FUNCTION_BLOCK FB_RecipeFactory_Test EXTENDS TcUnit.FB_TestSuite
VAR
    Factory : FB_RecipeFactory;
    Config  : ST_RecipeBuilder_Config;
END_VAR

Test_InjectsConfigProviderToAllBuilders();
Test_ReturnsCorrectBuilder();
Test_ReturnsZeroOnInvalidID();
Test_UpdatesConfigForAllBuilders();

METHOD Test_InjectsConfigProviderToAllBuilders
VAR_INST
    MockProvider : FB_MockConfigProvider;
END_VAR
VAR
    TestConfig       : ST_RecipeBuilder_Config;
    BuilderWings     : I_RecipeBuilder;
    BuilderFlaps     : I_RecipeBuilder;
    BuilderArona     : I_RecipeBuilder;
    BuilderCircle    : I_RecipeBuilder;
    BuilderRectangle : I_RecipeBuilder;
    
    iMockProvider    : I_GantryConfigProvider;
END_VAR
TEST('Test_InjectsConfigProviderToAllBuilders');

// 1. ARRANGE
// Rzutujemy instancję bloku na interfejs (aby kompilator wiedział, jak je porównywać)
iMockProvider := MockProvider;

// 2. ACT
Factory.InitializeFactory(Config := TestConfig, ConfigProvider := iMockProvider);

// Wyciągamy instancje z fabryki
BuilderWings     := Factory.GetBuilder(E_RecipeID.ePTPBorgoWings);
BuilderFlaps     := Factory.GetBuilder(E_RecipeID.ePTPBorgoFlaps);
BuilderArona     := Factory.GetBuilder(E_RecipeID.ePTPArona);
BuilderCircle    := Factory.GetBuilder(E_RecipeID.eNCICircle);
BuilderRectangle := Factory.GetBuilder(E_RecipeID.ePTPRectangle);

// 3. ASSERT
AssertTrue(Condition := (BuilderWings.ConfigProvider = iMockProvider),
           Message := 'BuilderWings nie otrzymal wstrzyknietego ConfigProvidera!');
AssertTrue(Condition := (BuilderFlaps.ConfigProvider = iMockProvider),
           Message := 'BuilderFlaps nie otrzymal wstrzyknietego ConfigProvidera!');
AssertTrue(Condition := (BuilderArona.ConfigProvider = iMockProvider),
           Message := 'BuilderArona nie otrzymal wstrzyknietego ConfigProvidera!');
AssertTrue(Condition := (BuilderCircle.ConfigProvider = iMockProvider),
           Message := 'BuilderCircle nie otrzymal wstrzyknietego ConfigProvidera!');
AssertTrue(Condition := (BuilderRectangle.ConfigProvider = iMockProvider),
           Message := 'BuilderRectangle nie otrzymal wstrzyknietego ConfigProvidera!');

TEST_FINISHED();
END_METHOD

METHOD Test_ReturnsCorrectBuilder
VAR
    BuilderWings     : I_RecipeBuilder;
    BuilderFlaps     : I_RecipeBuilder;
    BuilderArona     : I_RecipeBuilder;
    BuilderCircle    : I_RecipeBuilder; // Dodane!
    BuilderRectangle : I_RecipeBuilder; // Dodane!
END_VAR
TEST('Test_ReturnsCorrectBuilder');

// 1. ACT - Prosimy fabrykę o wszystkie wspierane przepisy
BuilderWings     := Factory.GetBuilder(E_RecipeID.ePTPBorgoWings);
BuilderFlaps     := Factory.GetBuilder(E_RecipeID.ePTPBorgoFlaps);
BuilderArona     := Factory.GetBuilder(E_RecipeID.ePTPArona);
BuilderCircle    := Factory.GetBuilder(E_RecipeID.eNCICircle);
BuilderRectangle := Factory.GetBuilder(E_RecipeID.ePTPRectangle);

// 2. ASSERT - Sprawdzamy, czy żaden z nich nie jest pusty (0)
AssertTrue(Condition := (BuilderWings <> 0), Message := 'Fabryka zwrocila 0 dla eBorgoWings!');
AssertTrue(Condition := (BuilderFlaps <> 0), Message := 'Fabryka zwrocila 0 dla eBorgoFlaps!');
AssertTrue(Condition := (BuilderArona <> 0), Message := 'Fabryka zwrocila 0 dla eArona!');
AssertTrue(Condition := (BuilderCircle <> 0), Message := 'Fabryka zwrocila 0 dla eCircle!');
AssertTrue(Condition := (BuilderRectangle <> 0), Message := 'Fabryka zwrocila 0 dla eRectangle!');

TEST_FINISHED();
END_METHOD

METHOD Test_ReturnsZeroOnInvalidID
VAR
    ReturnedBuilder : I_RecipeBuilder;
END_VAR


TEST('Test_ReturnsZeroOnInvalidID');

// Act - prosimy o eNone (ekran powitalny, bez wybranego programu)
ReturnedBuilder := Factory.GetBuilder(E_RecipeID.eNone);

// Assert - fabryka musi zwrócić 0
AssertTrue(Condition := (ReturnedBuilder = 0), 
           Message := 'Fabryka zwrocila interfejs zamiast 0 dla eNone!');

TEST_FINISHED();
END_METHOD

METHOD Test_UpdatesConfigForAllBuilders
VAR
    TestConfig : ST_RecipeBuilder_Config;
    
    BuilderWings : I_RecipeBuilder;
    BuilderFlaps : I_RecipeBuilder;
    BuilderArona : I_RecipeBuilder;
    
    // Zmienne pomocnicze, żeby obejść błąd kompilatora (odczyt właściwości)
    ActualConfigWings : ST_RecipeBuilder_Config;
    ActualConfigFlaps : ST_RecipeBuilder_Config;
    ActualConfigArona : ST_RecipeBuilder_Config;
END_VAR
TEST('Test_UpdatesConfigForAllBuilders');

// 1. ARRANGE - Tworzymy unikalną, testową konfigurację
TestConfig.PanelFrontLength := 999.0;
TestConfig.PanelHeight := 111.0;

// 2. ACT - Wrzucamy ją do fabryki, żeby rozesłała dalej
Factory.UpdateConfig(TestConfig);

// 3. Wyciągamy instancje z fabryki
BuilderWings := Factory.GetBuilder(E_RecipeID.ePTPBorgoWings);
BuilderFlaps := Factory.GetBuilder(E_RecipeID.ePTPBorgoFlaps);
BuilderArona := Factory.GetBuilder(E_RecipeID.ePTPArona);

// Zgrywamy konfigurację z właściwości interfejsów do zmiennych lokalnych
ActualConfigWings := BuilderWings.Config;
ActualConfigFlaps := BuilderFlaps.Config;
ActualConfigArona := BuilderArona.Config;

// 4. ASSERT - Sprawdzamy, czy wszyscy mają tę samą wartość
AssertEquals_REAL(Expected := 999.0, 
                  Actual := ActualConfigWings.PanelFrontLength, 
                  Delta := 0.01, 
                  Message := 'BuilderWings nie dostal nowej konfiguracji!');
                  
AssertEquals_REAL(Expected := 999.0, 
                  Actual := ActualConfigFlaps.PanelFrontLength, 
                  Delta := 0.01, 
                  Message := 'BuilderFlaps nie dostal nowej konfiguracji!');
                  
AssertEquals_REAL(Expected := 999.0, 
                  Actual := ActualConfigArona.PanelFrontLength, 
                  Delta := 0.01, 
                  Message := 'BuilderArona nie dostal nowej konfiguracji!');

TEST_FINISHED();
END_METHOD

END_FUNCTION_BLOCK

(* stored: Version 1.1.0.1, ProductVersion 3.1.4024.15
   POU FB_RecipeFactory_Test: Id {f26615a6-c66a-43dc-9573-a459ce1aeaeb}, SpecialFunc None
   Method Test_InjectsConfigProviderToAllBuilders: Id {d6313cf3-d5c8-436b-ba90-e789f33521a7}
   Method Test_ReturnsCorrectBuilder: Id {f4d0cc26-5c2a-4ddf-b356-c729fd5c6098}
   Method Test_ReturnsZeroOnInvalidID: Id {91b039b9-1372-48cc-8530-52ca18dfee07}
   Method Test_UpdatesConfigForAllBuilders: Id {4b2fa050-c8b8-4151-9cc7-69d180105cac} *)
